FUNCTION_BLOCK SpeedGauge (* Measures the linear speed from the rotary encoder count *)
  (* Standard: 61499-2 *)
  (* Version 0.2, 2003-12-04, JHC, Rockwell Automation, Renamed for better indexing. *)
  (* Version 0.1, 2002-11-05, JHC, Rockwell Automation, Corrected missing ST element in Algorithm REQ. *)
  (* Version 0.0, 2000-05-30, JHC, Rockwell Automation *)
  (* Compiler header: package fb.rt.benchmarks.cruisecontrol; *)
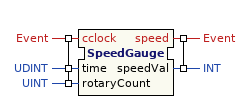
  EVENT_INPUT
    cclock WITH time, rotaryCount; (* 10ms tick *)
  END_EVENT
  EVENT_OUTPUT
    speed WITH speedVal;
  END_EVENT
  VAR_INPUT
    time : UDINT := 0; (* in us *)
    rotaryCount : UINT := 0; (* ranges from 0 to 1000 *)
  END_VAR
  VAR_OUTPUT
    speedVal : INT := 0; (* Output event qualifier *)
  END_VAR
  VAR
    prevCount : unsigned char := 0;
    prevTime : unsigned int := 0;
    count : unsigned short;
  END_VAR
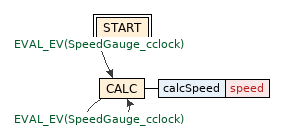
  EC_STATES
    START; (* Initial State *)
    CALC : calcSpeed -> speed;
  END_STATES
  EC_TRANSITIONS
    START TO CALC := EVAL_EV(SpeedGauge_cclock);
    CALC TO CALC := EVAL_EV(SpeedGauge_cclock);
  END_TRANSITIONS
  ALGORITHM calcSpeed IN ST:
if( VAL_OF_rotaryCount() >= prevCount){
    count= VAL_OF_rotaryCount() - prevCount;
}else{
    count= 1000 + VAL_OF_rotaryCount() - prevCount;
};

if( VAL_OF_speedVal() == 0) {
    VAL_OF_speedVal()= (count * 7012) / 10000;
}else{
    VAL_OF_speedVal()= (count * 7012) / 10000;
};

prevTime= VAL_OF_time();
prevCount= VAL_OF_rotaryCount();
  END_ALGORITHM
END_FUNCTION_BLOCK
